Fanuc KAREL source: V_GET_READ.kl

PROGRAM T
%NOLOCKGROUP
VAR
 v0 : STRING[40]
 v1 : INTEGER
 v2 : STRING[40]
 v3 : INTEGER
 v4 : INTEGER
BEGIN
 V_GET_READ(v0, v1, v2, v3, v4)
END T
